TEXTLIST TL_ACtype
  0 = 'Choose'
  1 = '0..10V'
  2 = '±10V'
  3 = '0..20mA'
  4 = '4..20mA'
   = ''
END_TEXTLIST

(* stored: Version 1.1.0.1, ProductVersion 3.1.4020.3
   TextList TL_ACtype: Id {44355528-9652-40ad-92a9-b4cda81a7a48} *)
